{attribute 'qualified_only'}
{attribute 'strict'}
TYPE ENUM_StageBrakeMode :
    // Defines when to send the brake disengage signal in FB_MotionStage
(
    IF_ENABLED, // Disengage brake when the motor is enabled
    IF_MOVING, // Disengage brake when the motor is moving
    NO_BRAKE // Do not change the brake state in FB_MotionStage
);
END_TYPE

(* stored: Version 1.1.0.1, ProductVersion 3.1.4022.18
   DUT ENUM_StageBrakeMode: Id {36cc1de7-1431-45ad-a25e-c90656daff0a} *)
